// TIA Portal V16 export
// export: Created 2022-11-17T15:49:42.8732389Z, ExportSetting WithDefaults, DisplayName Totally Integrated Automation Portal, DisplayVersion V16 Update 6, DisplayName TIA Portal Version Control Interface, DisplayVersion V16 Update 2, DisplayName TIA Portal Openness, DisplayVersion V16 Update 6, DisplayName SINAMICS Startdrive Advanced, DisplayVersion V16 Update 5, DisplayName SINAMICS Startdrive G130, G150, S120, S150, SINAMICS MV, S210, DisplayVersion V16 Update 5, DisplayName SINAMICS Startdrive G110M, G120, G120C, G120D, G120P, G115D, DisplayVersion V16 Update 5, DisplayName STEP 7 Professional, DisplayVersion V16 Update 6, DisplayName STEP 7 Safety, DisplayVersion V16, DisplayName WinCC Advanced, DisplayVersion V16 Update 6
DATA_BLOCK "DB215_ProgramData"   // DB215
TITLE = Program Data
{ S7_Optimized_Access := 'FALSE' }
VERSION : 0.1
// stored: AutoNumber false, IsOnlyStoredInLoadMemory false, IsWriteProtectedInAS false
   VAR RETAIN
      State_Initialization : UInt := 0;
      State_Setup : UInt := 0;
      InverterFault : Bool := FALSE;   // Inverter Fault (F) - Anomalia
      InverterAlarm : Bool := FALSE;   // Inverter Alarm (A) - Avviso
      Keylock : Bool := FALSE;   // Blocco tasti per utente
      ActiveRecipeMLC : Bool := FALSE;   // Multi-Level Control per la ricetta attiva
      Keylock2 : Bool := FALSE;   // Blocco tasti (StateAuto opp. blocco)
      RecipeModified : Bool := FALSE;
      RecipeSave : Bool := FALSE;
      LoadCellConst : Bool := TRUE;   // valore cella costante
      spare_5 : Bool := FALSE;
      spare_6 : Bool := FALSE;
      spare_7 : Bool := FALSE;
      spare_8 : Bool := FALSE;
      spare_9 : Bool := FALSE;
      spare_10 : Bool := FALSE;
      spare_11 : Bool := FALSE;
      spare_12 : Bool := FALSE;
      Offset_Pulses : Int := 0;   // NOT_USED
      Altimeter_Pulses : Int := 442;
      PhotDelay_Pulses : Int := 40;
      Reinforce_Pulses : Int := 0;
      TopFall_Pulses : Int := 134;
      ManRotStep : UInt := 0;
      RotSpeed : Int := 1770;
      CarSpeedUp : Int := 1396;
      CarSpeedDw : Int := 1396;
      Offset_cella : Int := 240;
      EncCarrDir : Int := -1;   // Direzione petalo carrello (1=av;-1=ind)
      EncCarrMax : Int := 603;   // Max altezza carrello (encoder)
      TiroObiettivo : UInt := 0;   // Tiro obiettivo (da chiamata FC300)
      ContaImpulsi : Int := 0;   // Contatore impulsi 20ms (OB30)
      MLC_HeightPulses : Int := 0;   // MLC_Height_Pulses
      MLC_Rounds : Int := 0;   // MLC_rounds
      LoadCellVal_1 : Int := 227;   // valore cella 1
      LoadCellVal_2 : Int := 227;   // valore cella 2
      PropArmMax : Int := 0;   // Costante proporzionalità corrisp. max freq. braccio
      PropCarrMax : Int := 0;   // Costante proporzionalità corrisp. max freq. carrello
      ValOffsetCella : Int := 10;   // Valore per offset cella durante il reset
      RoundTime : UInt := 4000;
      LastRoundTime : UInt := 2000;
      ReinforceTime : UInt := 0;   // [NOT USED]
      pTiro : Array[0..10] of UInt;
      iTiro : Array[0..10] of UInt;
   END_VAR
BEGIN
   pTiro[0] := 70;
   pTiro[1] := 60;
   pTiro[2] := 50;
   pTiro[3] := 45;
   pTiro[4] := 40;
   pTiro[5] := 35;
   pTiro[6] := 30;
   pTiro[7] := 25;
   pTiro[8..10] := 20;
   iTiro[0] := 70;
   iTiro[1] := 60;
   iTiro[2] := 50;
   iTiro[3] := 45;
   iTiro[4] := 40;
   iTiro[5] := 35;
   iTiro[6] := 30;
   iTiro[7] := 25;
   iTiro[8..10] := 20;
END_DATA_BLOCK
